TYPE ST_RmtLed :
STRUCT
	On: BOOL;
	InControl: BOOL;
	Hub1: BOOL;
	Hub2: BOOL;
	Alarm: BOOL;
END_STRUCT
END_TYPE

(* stored: Version 1.1.0.1, ProductVersion 3.1.4026.18
   DUT ST_RmtLed: Id {7502da17-a236-4910-8f33-5c83fe298163} *)
